PROGRAM PRG_Section_1
VAR
END_VAR

END_PROGRAM

(* stored: Version 1.1.0.1, ProductVersion 3.1.4022.12
   POU PRG_Section_1: Id {49021430-2479-452d-9fb0-1e4b70e05342}, SpecialFunc None *)
